SYSTEM TEST_TEXT (* Test of JTextPane-based components *)
  (* Standard: 61499-1 *)
  (* Version 0.0, 2004-06-20, JHC, Rockwell Automation *)
  APPLICATION APP1
  END_APPLICATION
  DEVICE DEV1 : FRAME_DEVICE
    RESOURCE WSTRINGS : PANEL_RESOURCE
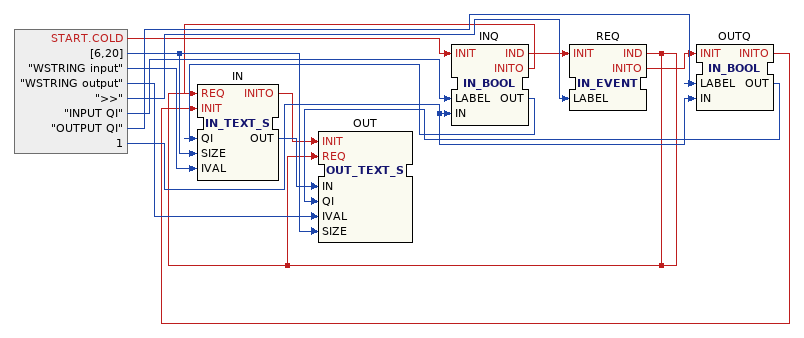
      FBS
        IN : IN_TEXT_S;
        OUT : OUT_TEXT_S;
        REQ : IN_EVENT;
        INQ : IN_BOOL;
        OUTQ : IN_BOOL;
      END_FBS
      EVENT_CONNECTIONS
        REQ.IND TO IN.REQ;
        IN.INITO TO OUT.INIT;
        INQ.IND TO IN.REQ;
        REQ.IND TO OUT.REQ;
        INQ.INITO TO REQ.INIT;
        REQ.INITO TO OUTQ.INIT;
        START.COLD TO INQ.INIT;
        OUTQ.INITO TO IN.INIT;
      END_CONNECTIONS
      DATA_CONNECTIONS
        INQ.OUT TO IN.QI;
        IN.OUT TO OUT.IN;
        OUTQ.OUT TO OUT.QI;
        [6,20] TO IN.SIZE;
        "WSTRING input" TO IN.IVAL;
        "WSTRING output" TO OUT.IVAL;
        [6,20] TO OUT.SIZE;
        ">>" TO REQ.LABEL;
        "INPUT QI" TO INQ.LABEL;
        "OUTPUT QI" TO OUTQ.LABEL;
        1 TO INQ.IN;
        1 TO OUTQ.IN;
      END_CONNECTIONS
    END_RESOURCE
    RESOURCE STRINGS : PANEL_RESOURCE
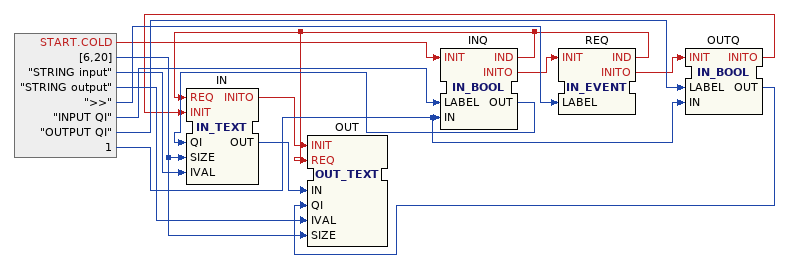
      FBS
        IN : IN_TEXT;
        OUT : OUT_TEXT;
        REQ : IN_EVENT;
        INQ : IN_BOOL;
        OUTQ : IN_BOOL;
      END_FBS
      EVENT_CONNECTIONS
        REQ.IND TO IN.REQ;
        IN.INITO TO OUT.INIT;
        INQ.IND TO IN.REQ;
        REQ.IND TO OUT.REQ;
        INQ.INITO TO REQ.INIT;
        REQ.INITO TO OUTQ.INIT;
        START.COLD TO INQ.INIT;
        OUTQ.INITO TO IN.INIT;
      END_CONNECTIONS
      DATA_CONNECTIONS
        INQ.OUT TO IN.QI;
        IN.OUT TO OUT.IN;
        OUTQ.OUT TO OUT.QI;
        [6,20] TO IN.SIZE;
        "STRING input" TO IN.IVAL;
        "STRING output" TO OUT.IVAL;
        [6,20] TO OUT.SIZE;
        ">>" TO REQ.LABEL;
        "INPUT QI" TO INQ.LABEL;
        "OUTPUT QI" TO OUTQ.LABEL;
        1 TO INQ.IN;
        1 TO OUTQ.IN;
      END_CONNECTIONS
    END_RESOURCE
  END_DEVICE
  DATA_CONNECTIONS (* parameter values *)
    [100,100,350,350] TO DEV1.BOUNDS;
    [2,1] TO DEV1.GRID;
  END_CONNECTIONS
END_SYSTEM
